{attribute addProperty BoxType "EL6201-0000-0017"}
{attribute addProperty Id "Slave_15A_DO0BIT10.125113Slave_15A_DO1BIT10.125114Slave_15A_DO2BIT10.125115Slave_15A_DO3BIT10.125116Slave_15B_DO0BIT10.125117Slave_15B_DO1BIT10.125118Slave_15B_DO2BIT10.125119Slave_15B_DO3BIT10.125120"}
{attribute addProperty CRC "1514304581"}
{attribute addProperty SizeInBites "8"}
{attribute addProperty SizeInBytes "1"}
TYPE Slave_15_Outputs_5A427445 :
STRUCT
	{attribute addProperty Name "Slave_15A_DO0"}
	Slave_15A_DO0 : BIT;
	{attribute addProperty Name "Slave_15A_DO1"}
	Slave_15A_DO1 : BIT;
	{attribute addProperty Name "Slave_15A_DO2"}
	Slave_15A_DO2 : BIT;
	{attribute addProperty Name "Slave_15A_DO3"}
	Slave_15A_DO3 : BIT;
	{attribute addProperty Name "Slave_15B_DO0"}
	Slave_15B_DO0 : BIT;
	{attribute addProperty Name "Slave_15B_DO1"}
	Slave_15B_DO1 : BIT;
	{attribute addProperty Name "Slave_15B_DO2"}
	Slave_15B_DO2 : BIT;
	{attribute addProperty Name "Slave_15B_DO3"}
	Slave_15B_DO3 : BIT;
END_STRUCT
END_TYPE

(* stored: Version 1.2.0.0, ProductVersion 3.1.4024.9
   DUT Slave_15_Outputs_5A427445: Id {32aea50d-eac2-42e1-a8a2-cc548f2f9411} *)
